FUNCTION_BLOCK WORD2WORD
  {SET_ATTRIBUTE(OpcUa, SERVICE)}
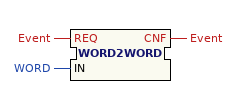
  EVENT_INPUT
    REQ;
  END_EVENT
  EVENT_OUTPUT
    CNF;
  END_EVENT
  VAR_INPUT
    IN : WORD;
  END_VAR
END_FUNCTION_BLOCK
